Universal Robots PolyScope program: sleeve test.urp

Program sleeve test (installation=default directory=/programs createdIn=5.14.5 lastSavedIn=5.14.5 robotSerialNumber=20236801216)
Calibrated DH parameters: a=[-0.000021, -0.748897, -0.28186, -0.00004, -0.000055, 0]; d=[0.236225, -424.082933, -1564.66872, 1988.95162, 0.159094, 0.153873]; alpha=[1.570844, 0.001002, 0.000337, 1.571488, -1.569996, 0]; deltaTheta=[0, -0.516316, 5.626292, 1.173211, 0.000001, 0]
InitVariablesNode
BeforeStart
  MoveJ speed 60 deg/s, acceleration 80 deg/s^2 (useActiveTCP=true) feature=Base
    Waypoint Waypoint_1: TCP in base x=891.483 y=352.796 z=387.488 mm, rx=2.3226 ry=2.0549 rz=0.0523 rad; joints [-187.011, -68.311, 93.408, 60.42, 0.058, -88.516] deg; TCP offset x=-5.49 y=-328 z=106.39 mm, rx=1.2092 ry=-1.2092 rz=1.2092 rad
  SafeHome (positionOptionType=SPEED_AND_ACCELERATION speed=1.047198 acceleration=1.396263 nextMotionTime=2)
  Set NoAction tcp=pretend_welder
  MoveJ speed 60 deg/s, acceleration 80 deg/s^2 (useActiveTCP=true) feature=Base
    Waypoint Waypoint_1: TCP in base x=891.483 y=352.796 z=387.488 mm, rx=2.3226 ry=2.0549 rz=0.0523 rad; joints [-187.011, -68.311, 93.408, 60.42, 0.058, -88.516] deg
    Waypoint Waypoint_2: TCP in base x=-839.646 y=463.039 z=9.516 mm, rx=0.8761 ry=-3.002 rz=-0.0791 rad; joints [-57.476, -54.43, 104.124, 24.159, 0.024, -76.85] deg
Robot Program (runOnlyOnce=true)
  MoveJ speed 60 deg/s, acceleration 80 deg/s^2 (useActiveTCP=true) feature=Base
    Waypoint Waypoint_2: TCP in base x=-839.646 y=463.039 z=9.516 mm, rx=0.8761 ry=-3.002 rz=-0.0791 rad; joints [-57.476, -54.43, 104.124, 24.159, 0.024, -76.85] deg
